Yaskawa INFORM job: OBROTK.JBI

/JOB
//NAME OBROTK
//POS
///NPOS 1,1,1,0,0,0
///TOOL 0
///POSTYPE PULSE
///PULSE
C00000=2000,-95440,-72516,0,38121,0
BC00000=23548,666204,788988
EC00000=-798156,1112951
//INST
///DATE 2024/03/05 20:04
///ATTR SC,RW
///GROUP1 RB1,BS1
///GROUP2 ST1
NOP
MOVJ C00000 BC00000 VJ=100.00  +MOVJ EC00000 VJ=100.00
END
